// TwinCAT 3 PLC project Untitled1
// ProgramVersion: 3.1.4026.12
// libraries:
//   Tc2_Standard, * (Beckhoff Automation GmbH)
//   Tc2_System, * (Beckhoff Automation GmbH)
//   Tc3_Module, * (Beckhoff Automation GmbH)
//   VisuDialogs, * (System)
// project tree:
//   DUTs/ E_Bedrijfstoestand.TcDUT, E_OpenDichtKlepState.TcDUT, E_RegelingState.TcDUT, E_RegelschuifState.TcDUT, E_PompState.TcDUT, E_Besturingsmodus.TcDUT
//   / FB_AlarmHandler.TcPOU, GlobalTextList.TcGTLO, PlcTask.TcTTO, Visualization Manager.TcVMO (not stored)
//   POUs/ControlLayer/ FB_Inmalen.TcPOU, FB_Regelingen.TcPOU, FB_Uitlaten.TcPOU, FB_Uitmalen.TcPOU
//   POUs/DeviceLayer/ FB_OpenDichtKlep.TcPOU, FB_Pomp.TcPOU, FB_Regelschuif_DG.TcPOU, FB_Regelschuif_AFO.TcPOU, ITF_OpenDichtKlep.TcIO, ITF_Regelschuif.TcIO, ITF_Pomp.TcIO
//   POUs/FieldLayer/OpenDichtKlep/ FB_SimulatedDigIn.TcPOU, FB_SimulatedDigOut.TcPOU, ITF_DigIn.TcIO, ITF_DigOut.TcIO
//   POUs/FieldLayer/Pomp/ FB_simulatedpompdigin.TcPOU, FB_simulatedpompdigout.TcPOU, FB_simulatiepompangout.TcPOU, ITF_pompangout.TcIO, ITF_pompdigin.TcIO, ITF_pompdigout.TcIO
//   POUs/FieldLayer/Regelschuif_AFO/ FB_SimulatedAnaIn_AFO.TcPOU, FB_SimulatedDigOutClose_AFO.TcPOU, FB_SimulatedDigOutOpen_AFO.TcPOU, ITF_Schuif_AnaIn_AFO.TcIO, ITF_Schuif_DigOutClose_AFO.TcIO, ITF_Schuif_DigOutOpen_AFO.TcIO
//   POUs/FieldLayer/Regelschuif_DG_1/ FB_SimulatedIn_DG.TcPOU, FB_SimulatedOutClose_DG.TcPOU, FB_SimulatedOutOpen_DG.TcPOU, ITF_Regelschuif_In_DG.TcIO, ITF_Regelschuif_OutClose_DG.TcIO, ITF_Regelschuif_OutOpen_DG.TcIO
//   POUs/ MAIN.TcPOU
//   VISUs/ Visualization.TcVIS
// real-time tasks:
//   TASK PlcTask: cycle T#10ms, priority 20, ADS port 350

CONFIGURATION Untitled1
    RESOURCE PLC ON TwinCAT3
        TASK PlcTask(INTERVAL := T#10ms, PRIORITY := 20);
        PROGRAM MAIN WITH PlcTask : MAIN;
    END_RESOURCE
END_CONFIGURATION

// ---- DUTs/E_Bedrijfstoestand.TcDUT
{attribute 'qualified_only'}
{attribute 'strict'}
{attribute 'to_string'}
TYPE E_Bedrijfstoestand :
(
	off := 0,
	manual,
	auto
);
END_TYPE

// ---- DUTs/E_OpenDichtKlepState.TcDUT
{attribute 'qualified_only'}
{attribute 'strict'}
{attribute 'to_string'}
TYPE E_OpenDichtKlepState :
(
	closed := 0,
	open,
	closing,
	opening,
	error
);
END_TYPE

// ---- DUTs/E_RegelingState.TcDUT
{attribute 'qualified_only'}
{attribute 'strict'}
{attribute 'to_string'}
TYPE E_RegelingState :
(
	uit := 0,
	polderpeil,
	debiet
);
END_TYPE

// ---- DUTs/E_RegelschuifState.TcDUT
{attribute 'qualified_only'}
{attribute 'strict'}
{attribute 'to_string'}
TYPE E_RegelschuifState :
(
	standby := 0,
	opening,
	closing,
	error
);
END_TYPE

// ---- DUTs/E_PompState.TcDUT
{attribute 'qualified_only'}
{attribute 'strict'}
{attribute 'to_string'}
TYPE E_PompState :
(
	off := 0,
	on,
	optoeren,
	aftoeren,
	error
);
END_TYPE

// ---- DUTs/E_Besturingsmodus.TcDUT
{attribute 'qualified_only'}
{attribute 'strict'}
{attribute 'to_string'}
TYPE E_Besturingsmodus :
(
	uitlaten := 0,
	uitmalen,
	inmalen
);
END_TYPE

// ---- POUs/DeviceLayer/ITF_OpenDichtKlep.TcIO
INTERFACE ITF_OpenDichtKlep

METHOD Close : BOOL
VAR_INPUT
END_VAR
END_METHOD

METHOD Open : BOOL
VAR_INPUT
END_VAR
END_METHOD

PROPERTY StateKlep : E_OpenDichtKlepState
GET
END_GET
SET
END_SET
END_PROPERTY

END_INTERFACE

// ---- POUs/DeviceLayer/ITF_Regelschuif.TcIO
INTERFACE ITF_Regelschuif

PROPERTY ActueelPosition : SINT
GET
END_GET
SET
END_SET
END_PROPERTY

METHOD RegelSchuifGoTo : SINT
VAR_INPUT
	regelschuifdoel : SINT;
END_VAR
END_METHOD

PROPERTY StateRegelSchuif : E_RegelschuifState
GET
END_GET
SET
END_SET
END_PROPERTY

END_INTERFACE

// ---- POUs/DeviceLayer/ITF_Pomp.TcIO
INTERFACE ITF_Pomp

PROPERTY ActueelToerental : INT
GET
END_GET
SET
END_SET
END_PROPERTY

METHOD PompGoTo : INT
VAR_INPUT
	toerental : INT;
END_VAR
END_METHOD

PROPERTY StatePomp : E_PompState
GET
END_GET
SET
END_SET
END_PROPERTY

END_INTERFACE

// ---- POUs/FieldLayer/OpenDichtKlep/ITF_DigIn.TcIO
INTERFACE ITF_DigIn

METHOD get : BOOL
VAR_INPUT
END_VAR
END_METHOD

END_INTERFACE

// ---- POUs/FieldLayer/OpenDichtKlep/ITF_DigOut.TcIO
INTERFACE ITF_DigOut

METHOD set : BOOL
VAR_INPUT
	state : BOOL;
END_VAR
END_METHOD

END_INTERFACE

// ---- POUs/FieldLayer/Pomp/ITF_pompangout.TcIO
INTERFACE ITF_pompangout

METHOD set : INT
VAR_INPUT
		state : INT;
END_VAR
END_METHOD

END_INTERFACE

// ---- POUs/FieldLayer/Pomp/ITF_pompdigin.TcIO
INTERFACE ITF_pompdigin

METHOD get : bool
VAR_INPUT
	state : BOOL;
END_VAR
END_METHOD

END_INTERFACE

// ---- POUs/FieldLayer/Pomp/ITF_pompdigout.TcIO
INTERFACE ITF_pompdigout

METHOD set : bool
VAR_INPUT
	state : BOOL;
END_VAR
END_METHOD

END_INTERFACE

// ---- POUs/FieldLayer/Regelschuif_AFO/ITF_Schuif_AnaIn_AFO.TcIO
INTERFACE ITF_Schuif_AnaIn_AFO

METHOD get : SINT
VAR_INPUT
END_VAR
END_METHOD

END_INTERFACE

// ---- POUs/FieldLayer/Regelschuif_AFO/ITF_Schuif_DigOutClose_AFO.TcIO
INTERFACE ITF_Schuif_DigOutClose_AFO

METHOD set : BOOL
VAR_INPUT
	state : BOOL;	
END_VAR
END_METHOD

END_INTERFACE

// ---- POUs/FieldLayer/Regelschuif_AFO/ITF_Schuif_DigOutOpen_AFO.TcIO
INTERFACE ITF_Schuif_DigOutOpen_AFO

METHOD set : BOOL
VAR_INPUT
	state : BOOL;
END_VAR
END_METHOD

END_INTERFACE

// ---- POUs/FieldLayer/Regelschuif_DG_1/ITF_Regelschuif_In_DG.TcIO
INTERFACE ITF_Regelschuif_In_DG

METHOD get : SINT
VAR_INPUT
END_VAR
END_METHOD

END_INTERFACE

// ---- POUs/FieldLayer/Regelschuif_DG_1/ITF_Regelschuif_OutClose_DG.TcIO
INTERFACE ITF_Regelschuif_OutClose_DG

METHOD set : BOOL
VAR_INPUT
	state : BOOL;	
END_VAR
END_METHOD

END_INTERFACE

// ---- POUs/FieldLayer/Regelschuif_DG_1/ITF_Regelschuif_OutOpen_DG.TcIO
INTERFACE ITF_Regelschuif_OutOpen_DG

METHOD set : BOOL
VAR_INPUT
	state : BOOL;
END_VAR
END_METHOD

END_INTERFACE

// ---- POUs/MAIN.TcPOU
PROGRAM MAIN
VAR
	alarms  : FB_AlarmHandler;
	
	// Start digin digout van appeltjes
	digIn_V2012_1 : FB_SimulatedDigIn;
	digIn_V2012_2 : FB_SimulatedDigIn;
	digOut_V2012 : FB_SimulatedDigOut;
	
	digIn_V2014_1 : FB_SimulatedDigIn;
	digIn_V2014_2 : FB_SimulatedDigIn;
	digOut_V2014 : FB_SimulatedDigOut;
	
	digIn_V2021_1 : FB_SimulatedDigIn;
	digIn_V2021_2 : FB_SimulatedDigIn;
	digOut_V2021 : FB_SimulatedDigOut;
	
	digIn_V2023_1 : FB_SimulatedDigIn;
	digIn_V2023_2 : FB_SimulatedDigIn;
	digOut_V2023 : FB_SimulatedDigOut;
	
	digIn_V2024_1 : FB_SimulatedDigIn;
	digIn_V2024_2 : FB_SimulatedDigIn;
	digOut_V2024 : FB_SimulatedDigOut;
	
	digIn_V2025_1 : FB_SimulatedDigIn;
	digIn_V2025_2 : FB_SimulatedDigIn;
	digOut_V2025 : FB_SimulatedDigOut;
	
	digIn_V2026_1 : FB_SimulatedDigIn;
	digIn_V2026_2 : FB_SimulatedDigIn;
	digOut_V2026 : FB_SimulatedDigOut;
	// Einde digin digout van appeltjes
	
	// Start digin digout van AFO
	digOutOpeningV2013 : FB_SimulatedDigOutOpen_AFO;
	digOutClosingV2013 :FB_SimulatedDigOutClose_AFO;
	AnaInV2013 : FB_SimulatedAnaIn_AFO;
	
	digOutOpeningV2022 : FB_SimulatedDigOutOpen_AFO;
	digOutClosingV2022 :FB_SimulatedDigOutClose_AFO;
	AnaInV2022 : FB_SimulatedAnaIn_AFO;
	
	AFOTarget : SINT := 20; 
	AFOTarget2 : SINT; 
	// Einde digin digout van AFO

	//DG
	OutOpeningV2013 : FB_SimulatedOutOpen_DG;
	OutClosingV2013 :FB_SimulatedOutClose_DG;
	InV2013 : FB_SimulatedIn_DG;
	
	OutOpeningV2022 : FB_SimulatedOutOpen_DG;
	OutClosingV2022 :FB_SimulatedOutClose_DG;
	InV2022 : FB_SimulatedIn_DG;
	//DG

	// Start digin digout van queens of harts
	digoutP2011 :FB_simulatedpompdigout;
	digoutP2021 :FB_simulatedpompdigout;
	diginP2011 : FB_simulatedpompdigin;
	diginP2021 : FB_simulatedpompdigin;
	AnaoutP2011 : FB_simulatiepompangout;
	AnaoutP2021 : FB_simulatiepompangout;
	
	
	// einde digin digout van queens of harts
	V2012 : FB_OpenDichtKlep(tag := 'V2012', DigInClosed := digIn_V2012_1, DigInOpened := digIn_V2012_2, DigOut := digOut_V2012);
	V2014 : FB_OpenDichtKlep(tag := 'V2014', DigInClosed := digIn_V2014_1, DigInOpened := digIn_V2014_2, DigOut := digOut_V2014);
	V2021 : FB_OpenDichtKlep(tag := 'V2021', DigInClosed := digIn_V2021_1, DigInOpened := digIn_V2021_2, DigOut := digOut_V2021);
	V2023 : FB_OpenDichtKlep(tag := 'V2023', DigInClosed := digIn_V2023_1, DigInOpened := digIn_V2023_2, DigOut := digOut_V2023);
	V2024 : FB_OpenDichtKlep(tag := 'V2024', DigInClosed := digIn_V2024_1, DigInOpened := digIn_V2024_2, DigOut := digOut_V2024);  
	V2025 : FB_OpenDichtKlep(tag := 'V2025', DigInClosed := digIn_V2025_1, DigInOpened := digIn_V2025_2, DigOut := digOut_V2025);  
	V2026 : FB_OpenDichtKlep(tag := 'V2026', DigInClosed := digIn_V2026_1, DigInOpened := digIn_V2026_2, DigOut := digOut_V2026);  
	
	V2013_AFO : FB_Regelschuif_AFO(tag := 'V2013', DigOutOpening := digOutOpeningV2013, DigOutClosing := digOutClosingV2013, AnaInPosition := AnaInV2013);
	V2022_AFO : FB_Regelschuif_AFO(tag := 'V2022', DigOutOpening := digOutOpeningV2022, DigOutClosing := digOutClosingV2022, AnaInPosition := AnaInV2022);
	
	V2013_DG : FB_Regelschuif_DG(tag := 'V2013', OutputOpen := OutOpeningV2013, OutputClose := OutClosingV2013, SchuifInput := InV2013);
	V2022_DG : FB_Regelschuif_DG(tag := 'V2022', OutputOpen := OutOpeningV2022, OutputClose := OutClosingV2022, SchuifInput := InV2022);
	
	P2011 : FB_Pomp(tag:= 'P2011',DigOutOn:=digoutP2011,Diginon:=diginP2011, Anaouttoerental:=AnaoutP2011);
	P2021 : FB_Pomp(tag:= 'P2021',DigOutOn:=digoutP2021,Diginon:=diginP2021, Anaouttoerental:=AnaoutP2021);
	
	Regelingen : FB_Regelingen;
	
	ControllerInmalen : FB_Inmalen(OpenDichtKlepV2012 := V2012,
								   OpenDichtKlepV2014 := V2014,
								   OpenDichtKlepV2021 := V2021, 
								   OpenDichtKlepV2023 := V2023, 
								   OpenDichtKlepV2024 := V2024,
								   OpenDichtKlepV2025 := V2025,
								   OpenDichtKlepV2026 := V2026,
								   RegelschuifV2013_AFO := V2013_AFO,
								   RegelschuifV2022_AFO := V2022_AFO,
								   RegelschuifV2013_DG := V2013_DG,
								   RegelschuifV2022_DG := V2022_DG,
								   PompP2011 := P2011,
								   PompP2021 := P2021 );
								   
	ControllerUitmalen : FB_Uitmalen(OpenDichtKlepV2012 := V2012,
								   OpenDichtKlepV2014 := V2014,
								   OpenDichtKlepV2021 := V2021, 
								   OpenDichtKlepV2023 := V2023, 
								   OpenDichtKlepV2024 := V2024,
								   OpenDichtKlepV2025 := V2025,
								   OpenDichtKlepV2026 := V2026,
								   RegelschuifV2013_AFO := V2013_AFO,
								   RegelschuifV2022_AFO := V2022_AFO,
								   RegelschuifV2013_DG := V2013_DG,
								   RegelschuifV2022_DG := V2022_DG,
								   PompP2021 := P2021,
								   PompP2011 := P2011 );
								   
	ControllerUitlaten: FB_Uitlaten(OpenDichtKlepV2012:= V2012,
									OpenDichtKlepV2021:=V2021,
									OpenDichtKlepV2023:=V2023,
									OpenDichtKlepV2024:=V2024,
									V2013_DG:=V2013_DG,
									V2022_DG:=V2022_DG,
									V2013_AFO:=V2013_AFO,
									V2022_AFO:=V2022_AFO,
									Pomp2011:= P2011,
									Pomp2021:= P2021);					   
	ManToerental2011: INT;
	ManToerental2021: INT;
	
	ManKlepstand2013_DG: SINT;
	ManKlepstand2022_DG: SINT;
END_VAR

digIn_V2012_1();
digIn_V2012_2();
digOut_V2012();

digIn_V2021_1();
digIn_V2021_2();
digOut_V2021();

digIn_V2023_1();
digIn_V2023_2();
digOut_V2023();

digIn_V2024_1();
digIn_V2024_2();
digOut_V2024();

digIn_V2025_1();
digIn_V2025_2();
digOut_V2025();

digIn_V2026_1();
digIn_V2026_2();
digOut_V2026();

digIn_V2014_1();
digIn_V2014_2();
digOut_V2014();

V2012();
V2014();
V2021();
V2023();
V2024();
V2025();
V2026();
//End  function kleppen appeltjes

P2021();
P2011();
P2011.PompGoToManual(ManToerental2011);
P2021.PompGoToManual(ManToerental2021);


Regelingen ();
ControllerInmalen ();
ControllerUitmalen ();
ControllerUitlaten();

//AFO
digOutOpeningV2013();
digOutClosingV2013();
AnaInV2013();
V2013_AFO();
V2013_AFO.RegelSchuifGoTo(AFOTarget); // voor handmatige test
digOutOpeningV2022();
digOutClosingV2022();
AnaInV2022();
V2022_AFO();
V2022_AFO.RegelSchuifGoTo(AFOTarget2); // voor handmatige test

//DG
V2013_DG();
V2013_DG.RegelSchuifGoToManual(ManKlepstand2013_DG);
V2022_DG();
V2022_DG.RegelSchuifGoToManual(ManKlepstand2022_DG);

END_PROGRAM

// ---- FB_AlarmHandler.TcPOU
FUNCTION_BLOCK FB_AlarmHandler
VAR
END_VAR

METHOD Append : BOOL
VAR_INPUT
	tag : STRING;
	msg : STRING;
END_VAR
VAR
	str : STRING;
END_VAR
str := CONCAT(tag, ': ');
str := CONCAT(str, msg);
ADSLOGSTR(msgCtrlMask := ADSLOG_MSGTYPE_WARN OR ADSLOG_MSGTYPE_MSGBOX, msgFmtStr := '%s!', strArg := str);
END_METHOD

END_FUNCTION_BLOCK

// ---- POUs/FieldLayer/OpenDichtKlep/FB_SimulatedDigIn.TcPOU
FUNCTION_BLOCK FB_SimulatedDigIn IMPLEMENTS ITF_DigIn
VAR
	internalState : BOOL;
END_VAR

METHOD get : BOOL
VAR_INPUT
END_VAR
get := internalState;
END_METHOD

END_FUNCTION_BLOCK

// ---- POUs/FieldLayer/OpenDichtKlep/FB_SimulatedDigOut.TcPOU
FUNCTION_BLOCK FB_SimulatedDigOut IMPLEMENTS ITF_DigOut
VAR
	internalState : BOOL := FALSE;
END_VAR

METHOD set : BOOL
VAR_INPUT
	state : BOOL;
END_VAR
internalState := state;
END_METHOD

END_FUNCTION_BLOCK

// ---- POUs/FieldLayer/Regelschuif_AFO/FB_SimulatedDigOutOpen_AFO.TcPOU
FUNCTION_BLOCK FB_SimulatedDigOutOpen_AFO IMPLEMENTS ITF_Schuif_DigOutOpen_AFO
VAR
	internalState : BOOL := FALSE;
END_VAR

METHOD set : BOOL
VAR_INPUT
	state : BOOL;
END_VAR
internalState := state;
END_METHOD

END_FUNCTION_BLOCK

// ---- POUs/FieldLayer/Regelschuif_AFO/FB_SimulatedDigOutClose_AFO.TcPOU
FUNCTION_BLOCK FB_SimulatedDigOutClose_AFO IMPLEMENTS ITF_Schuif_DigOutClose_AFO
VAR
	internalState : BOOL := FALSE;
END_VAR

{warning 'Add method implementation '}
METHOD set : BOOL
VAR_INPUT
	state : BOOL;
END_VAR
internalState := state;
END_METHOD

END_FUNCTION_BLOCK

// ---- POUs/FieldLayer/Regelschuif_AFO/FB_SimulatedAnaIn_AFO.TcPOU
FUNCTION_BLOCK FB_SimulatedAnaIn_AFO IMPLEMENTS ITF_Schuif_AnaIn_AFO

VAR
	internalState : sint;
END_VAR

{warning 'Add method implementation '}
METHOD get : SINT
get := internalState;
END_METHOD

END_FUNCTION_BLOCK

// ---- POUs/FieldLayer/Regelschuif_DG_1/FB_SimulatedOutOpen_DG.TcPOU
FUNCTION_BLOCK FB_SimulatedOutOpen_DG IMPLEMENTS ITF_Regelschuif_OutOpen_DG
VAR
	internalState : BOOL := FALSE;
END_VAR

METHOD set : BOOL
VAR_INPUT
	state : BOOL;
END_VAR
internalState := state;
END_METHOD

END_FUNCTION_BLOCK

// ---- POUs/FieldLayer/Regelschuif_DG_1/FB_SimulatedOutClose_DG.TcPOU
FUNCTION_BLOCK FB_SimulatedOutClose_DG IMPLEMENTS ITF_Regelschuif_OutClose_DG
VAR
	internalState : BOOL := FALSE;
END_VAR

{warning 'Add method implementation '}
METHOD set : BOOL
VAR_INPUT
	state : BOOL;
END_VAR
internalState := state;
END_METHOD

END_FUNCTION_BLOCK

// ---- POUs/FieldLayer/Regelschuif_DG_1/FB_SimulatedIn_DG.TcPOU
FUNCTION_BLOCK FB_SimulatedIn_DG IMPLEMENTS ITF_Regelschuif_IN_DG

VAR
	internalState : sint;
END_VAR

{warning 'Add method implementation '}
METHOD get : SINT
get := internalState;
END_METHOD

END_FUNCTION_BLOCK

// ---- POUs/FieldLayer/Pomp/FB_simulatedpompdigout.TcPOU
FUNCTION_BLOCK FB_simulatedpompdigout IMPLEMENTS ITF_pompdigout
VAR
	internalState:BOOL;
END_VAR

{warning 'Add method implementation '}
METHOD set : BOOL
VAR_INPUT
	state	: BOOL;
END_VAR
internalState := state;
END_METHOD

END_FUNCTION_BLOCK

// ---- POUs/FieldLayer/Pomp/FB_simulatedpompdigin.TcPOU
FUNCTION_BLOCK FB_simulatedpompdigin IMPLEMENTS ITF_pompdigin
VAR
	internalState : bool;
END_VAR

{warning 'Add method implementation '}
METHOD get : BOOL
VAR_INPUT
	state	: BOOL;
END_VAR
get := internalState;
END_METHOD

END_FUNCTION_BLOCK

// ---- POUs/FieldLayer/Pomp/FB_simulatiepompangout.TcPOU
FUNCTION_BLOCK FB_simulatiepompangout IMPLEMENTS ITF_pompangout

VAR
		internalState : int;
END_VAR

METHOD set : INT
VAR_INPUT
	state	: INT;
END_VAR
internalState := state;
END_METHOD

END_FUNCTION_BLOCK

// ---- POUs/DeviceLayer/FB_OpenDichtKlep.TcPOU
FUNCTION_BLOCK FB_OpenDichtKlep IMPLEMENTS ITF_OpenDichtKlep
VAR
    tagName : STRING;
    inputOpen : ITF_DigIn;
	inputClosed : ITF_DigIn;
	output : ITF_DigOut;
	
	feedbackOpen : BOOL := FALSE;
	feedbackClosed : BOOL := FALSE;
	feedbackError : BOOL := FALSE;
	
	manOpen : BOOL := FALSE;
	manClose : BOOL := FALSE;

	currentMode : E_Bedrijfstoestand := E_Bedrijfstoestand.off;
	currentState : E_OpenDichtKlepState := E_OpenDichtKlepState.closed;
	expectedState : E_OpenDichtKlepState := E_OpenDichtKlepState.closed;
	
	timeOut : TON;
	errorTrigger : R_TRIG;
	

END_VAR

//check if currentmode = off and set klep closed
IF currentMode = E_Bedrijfstoestand.off THEN
	output.set(FALSE);
	expectedState := E_OpenDichtKlepState.closed;
END_IF

//check if currentmode = manual and give klep a state
IF currentMode = E_Bedrijfstoestand.manual THEN
	IF manOpen THEN
		openManual();
		manOpen:= FALSE;
	END_IF
	IF manClose THEN
		closeManual();
		manClose:= FALSE;
	END_IF
END_IF

//control witch feedback button in pressed
feedbackOpen := inputOpen.get() AND NOT inputClosed.get();
feedbackClosed := inputClosed.get() AND NOT inputOpen.get();
feedbackError := inputClosed.get() AND inputOpen.get();

//set timer for error
timeOut(IN := NOT(expectedState = currentState), PT := T#5S);
errorTrigger(CLK := (timeOut.Q OR feedbackError));

//check if error is active
IF errorTrigger.Q THEN
	currentState := E_OpenDichtKlepState.error;
	main.alarms.append(tag := tagName, msg := 'Klepstoring gedetecteerd');
END_IF

//set state of klep based on feedback buttons
IF feedbackClosed THEN
	currentState := E_OpenDichtKlepState.closed;
ELSIF NOT(currentState = E_OpenDichtKlepState.error) AND expectedState = E_OpenDichtKlepState.closed THEN
	currentState := E_OpenDichtKlepState.closing;
ELSIF feedbackOpen THEN
	currentState := E_OpenDichtKlepState.open;
ELSIF NOT(currentState = E_OpenDichtKlepState.error)AND expectedState = E_OpenDichtKlepState.open THEN
	currentState := E_OpenDichtKlepState.opening;
END_IF

METHOD close : BOOL
VAR_INPUT
END_VAR
IF currentMode = E_Bedrijfstoestand.auto THEN
	output.set(FALSE);
	expectedState := E_OpenDichtKlepState.closed;
	close := TRUE;
ELSE
	close := FALSE;
END_IF
END_METHOD

METHOD closeManual : BOOL
VAR_INPUT
END_VAR
IF currentMode = E_Bedrijfstoestand.manual THEN
	output.set(FALSE);
	expectedState := E_OpenDichtKlepState.closed;
	closeManual := TRUE;
ELSE
	closeManual := FALSE;
END_IF
END_METHOD

METHOD FB_init : BOOL
VAR_INPUT
	bInitRetains : BOOL; // if TRUE, the retain variables are initialized (warm start / cold start)
	bInCopyCode : BOOL;  // if TRUE, the instance afterwards gets moved into the copy code (online change)
	tag : STRING;
	DigInClosed : ITF_DigIn;
	DigInOpened : ITF_DigIn;
	DigOut : ITF_DigOut;
END_VAR
tagname := tag;
inputClosed := DigInClosed;
inputOpen := DigInOpened;
output := DigOut;
END_METHOD

METHOD open : BOOL
VAR_INPUT
END_VAR
IF currentMode = E_Bedrijfstoestand.auto THEN
	output.set(TRUE);
	expectedState := E_OpenDichtKlepState.open;
	open := TRUE;
ELSE
	open := FALSE;
END_IF
END_METHOD

METHOD openManual : BOOL
VAR_INPUT
END_VAR
IF currentMode = E_Bedrijfstoestand.manual THEN
	output.set(TRUE);
	expectedState := E_OpenDichtKlepState.open;
	openManual := TRUE;
ELSE
	openManual := FALSE;
END_IF
END_METHOD

PROPERTY StateKlep : E_OpenDichtKlepState
GET
StateKlep := currentState;
END_GET
SET
END_SET
END_PROPERTY

END_FUNCTION_BLOCK

// ---- POUs/DeviceLayer/FB_Regelschuif_AFO.TcPOU
FUNCTION_BLOCK FB_Regelschuif_AFO IMPLEMENTS ITF_Regelschuif
VAR
	tagName : STRING;
	outputOpen : ITF_Schuif_DigOutOpen_AFO;
	outputClose : ITF_Schuif_DigOutClose_AFO;
	inputPosition : ITF_Schuif_AnaIn_AFO;

	currentMode : E_Bedrijfstoestand := E_Bedrijfstoestand.off;
	currentState : E_RegelschuifState := E_RegelschuifState.standby;
	expectedState : E_RegelschuifState := E_RegelschuifState.standby;
	
	feedbackPosition : SINT;
	
	timeOut : TON;
	errorTrigger : R_TRIG;
	positie : SINT;
	secondTimerRun : BOOL;
	secondTimerTrigger : R_TRIG;
	
	timerrunt: BOOL:=1;
	waitExtraMinute: BOOL;
	minuteTimer : TON;
	doubleMinuteTimer : TON;
	secondTimer : TON;
	
	veranderingsMargeError : SINT := 3;
	OldPosition: SINT;
	regelschuifMargin: SINT := 3;
END_VAR

// Als de mode is uit dan worden de outputs false geset 
IF currentMode = E_Bedrijfstoestand.off THEN
	outputOpen.set(FALSE);
	outputClose.set(FALSE);
END_IF

// De feedback positie staat hiet zodat we de waardes kunnen veranderen
feedbackPosition := inputPosition.get();
ActueelPosition := inputPosition.get();

// Dit is de timer om te checken of er een error moet zijn 
timeOut(IN :=(StateRegelSchuif <> E_RegelschuifState.standby) AND NOT timeOut.Q, PT := T#30S);
errorTrigger(CLK := timeOut.Q);

IF errorTrigger.Q THEN
	IF (ActueelPosition < (OldPosition + veranderingsMargeError)) AND StateRegelSchuif = E_RegelschuifState.opening THEN
		StateRegelSchuif := E_RegelschuifState.error;
		main.alarms.append(tag := tagName, msg := 'Schuifstoring gedetecteerd, te langzaam openen');
	END_IF
	IF (ActueelPosition > (OldPosition - veranderingsMargeError)) AND StateRegelSchuif = E_RegelschuifState.closing THEN
		StateRegelSchuif := E_RegelschuifState.error;
		main.alarms.append(tag := tagName, msg := 'Schuifstoring gedetecteerd, te langzaam sluiten');
	END_IF
	IF StateRegelSchuif = E_RegelschuifState.error AND (ActueelPosition > (OldPosition + veranderingsMargeError)) THEN
		StateRegelSchuif := E_RegelschuifState.opening;
		ELSIF StateRegelSchuif = E_RegelschuifState.error AND (ActueelPosition < (OldPosition - veranderingsMargeError)) THEN
			StateRegelSchuif := E_RegelschuifState.closing;
	END_IF
	OldPosition := ActueelPosition;
END_IF

expectedState := StateRegelSchuif;

PROPERTY ActueelPosition : SINT
GET
ActueelPosition := feedbackPosition;
END_GET
SET
feedbackPosition := ActueelPosition;
END_SET
END_PROPERTY

//FB_Init is always available implicitly and it is used primarily for initialization.
//The return value is not evaluated. For a specific influence, you can also declare the
//methods explicitly and provide additional code there with the standard initialization
//code. You can evaluate the return value.
METHOD FB_Init: BOOL
VAR_INPUT
    bInitRetains: BOOL; // TRUE: the retain variables are initialized (reset warm / reset cold)
    bInCopyCode: BOOL;  // TRUE: the instance will be copied to the copy code afterward (online change)   
	tag : STRING;
	DigOutOpening : ITF_Schuif_DigOutOpen_AFO;
	DigOutClosing : ITF_Schuif_DigOutClose_AFO;
	AnaInPosition : ITF_Schuif_AnaIn_AFO;
END_VAR
tagname := tag;
outputOpen := DigOutOpening;
outputClose := DigOutClosing;
inputPosition := AnaInPosition;
END_METHOD

METHOD RegelSchuifGoTo : SINT
VAR	
	checkPositions : BOOL;
	currentstatet: E_RegelschuifState;
	secondTriggerTrigger: BOOL;
END_VAR
VAR_INPUT
	regelschuifdoel : SINT;
END_VAR
minuteTimer(IN:= timerrunt,PT:= T#10S);
doubleMinuteTimer(IN:= waitExtraMinute,PT:= T#10S); // tweede timer om een extra minuut te wachten na pulse maar niet langer te wachten met scannen

// dit is zodat het gefaseerd gaat een pulse per sec sturen
secondTimer(IN:= secondTimerRun,PT:= T#2S); // pulse lengte langer ivm testen

IF currentMode = E_Bedrijfstoestand.off THEN
	regelschuifdoel := ActueelPosition;
END_IF

IF minuteTimer.Q THEN
	
	IF ActueelPosition >= (regelschuifdoel - regelschuifMargin) AND ActueelPosition <= (regelschuifdoel + regelschuifMargin) THEN // huidige positie is correct binnen marge
		StateRegelSchuif := E_RegelschuifState.standby;
		outputOpen.set(FALSE); // set outputs naar 0 als extra backup
		outputClose.set(FALSE);
	
	END_IF
	
	IF ActueelPosition > (regelschuifdoel + regelschuifMargin) AND waitExtraMinute = FALSE THEN // huidige positie is te hoog
		IF stateRegelschuif <> E_RegelschuifState.error THEN
			StateRegelSchuif := E_RegelschuifState.closing;
		END_IF
		// voor de pulse		
		outputOpen.set(FALSE);
		outputClose.set(TRUE);
		secondTimerRun := TRUE; // start pulse time
		waitExtraMinute := TRUE; // wacht een minuut extra als er een pulse is gestuurd
	END_IF

	IF ActueelPosition < (regelschuifdoel - regelschuifMargin) AND waitExtraMinute = FALSE THEN // huidige positie is te laag
		IF stateRegelschuif <> E_RegelschuifState.error THEN
			StateRegelSchuif := E_RegelschuifState.opening;
		END_IF
		// voor de pulse
		outputClose.set(FALSE);
		outputOpen.set(TRUE);
		secondTimerRun := TRUE; // start pulse time
		waitExtraMinute := TRUE;
	END_IF
	timerrunt := 0; // reset timer
ELSIF waitExtraMinute = FALSE OR doubleMinuteTimer.Q THEN 
	waitExtraMinute := FALSE;
	timerrunt := 1; //reser reset timer
END_IF

// pulse timer structuur
IF secondTimer.Q THEN
	outputClose.set(FALSE);
	outputOpen.set(FALSE);
	secondTimerRun := FALSE;
END_IF

positie := regelschuifdoel;
END_METHOD

PROPERTY StateRegelSchuif : E_RegelschuifState
GET
StateRegelschuif := currentState;
END_GET
SET
currentstate:= StateRegelSchuif;
END_SET
END_PROPERTY

END_FUNCTION_BLOCK

// ---- POUs/DeviceLayer/FB_Regelschuif_DG.TcPOU
FUNCTION_BLOCK FB_Regelschuif_DG IMPLEMENTS ITF_Regelschuif
VAR
	TagName: STRING;
	
	OpenSchuif: ITF_Regelschuif_OutOpen_DG;
	SluitSchuif: ITF_Regelschuif_OutClose_DG;
	InputSchuif: ITF_Regelschuif_In_DG;
	
	CurrentMode: E_Bedrijfstoestand:= E_Bedrijfstoestand.off;
	currentState : E_RegelschuifState := E_RegelschuifState.standby;
	expectedState : E_RegelschuifState := E_RegelschuifState.standby;
	
	feedbackposition: SINT;
	VorigePosition: SINT;
	Marge : SINT := 2;
	schuifverandering: SINT:= 1;
	Doelschuif: SINT;
	DoelschuifAuto : SINT;
	VorigDoel: SINT;
	
	PulseTimer: TON;
	StartPulse: BOOL;
	Pulsetrigger: R_TRIG;
	
	OptelTimer: TON;
	StartOptel: BOOL;
	
	error_Trigger: R_TRIG;
	ErrorTimer: TON;
	SchuifsturingOpen: BOOL;
	SchuifsturingSluit: BOOL;
	SchuifStandby: BOOL;
END_VAR

//Als de schuif uit staat stopt de regelschuif met openen of sluiten
IF CurrentMode = E_Bedrijfstoestand.off THEN
	Currentstate:= E_Regelschuifstate.standby;
END_IF

//De actuele positie van de schuif wordt geupdate
ActueelPosition:= Feedbackposition;

ErrorTimer(IN:= Currentstate <> E_Regelschuifstate.standby AND NOT ErrorTimer.Q ,PT:= T#5S);
error_Trigger(CLK:= ErrorTimer.Q);

PulseTimer(IN:=StartPulse AND NOT PulseTimer.Q ,PT:= T#10S);
Pulsetrigger(CLK:= Pulsetimer.Q);
IF (Currentmode <> E_Bedrijfstoestand.off) AND NOT Pulsetimer.Q THEN
	Startpulse:= 1;
END_IF

IF Currentmode = E_Bedrijfstoestand.off THEN
	SchuifsturingOpen := FALSE;
	SchuifsturingSluit := FALSE;
	Openschuif.set(FALSE);
	SluitSchuif.set(FALSE);
END_IF

IF (Pulsetrigger.Q) OR ((Doelschuif <> Vorigdoel)
AND CurrentMode = E_Bedrijfstoestand.manual) THEN
	Startpulse:= 0;
	IF (Doelschuif < Feedbackposition) THEN
		SchuifsturingOpen := FALSE;
		SchuifsturingSluit := TRUE;
	END_IF	
	IF (Doelschuif > Feedbackposition) THEN
		SchuifsturingOpen := TRUE;
		SchuifsturingSluit := FALSE;
	END_IF
	StartPulse:= 1;
	Vorigdoel:= Doelschuif;
END_IF

IF Feedbackposition = 100 OR Feedbackposition = 0 THEN;
	Currentstate := E_RegelschuifState.standby;
	Schuifsturing();
ELSIF (Doelschuif < Feedbackposition) THEN
	Currentstate := E_RegelschuifState.closing;
ELSIF (Doelschuif > Feedbackposition) THEN
	Currentstate := E_RegelschuifState.opening;
ELSIF (DoelschuifAuto < Feedbackposition) THEN
	Currentstate := E_RegelschuifState.closing;
ELSIF (DoelschuifAuto > Feedbackposition) THEN
	Currentstate := E_RegelschuifState.opening;
END_IF

IF SchuifsturingSluit OR SchuifsturingOpen THEN
	Schuifsturing();
END_IF


IF (Pulsetrigger.Q)
AND CurrentMode = E_Bedrijfstoestand.auto THEN
	Startpulse:= 0;
	IF (DoelschuifAuto < Feedbackposition) THEN
		SchuifsturingOpen := FALSE;
		SchuifsturingSluit := TRUE;
	END_IF	
	IF (DoelschuifAuto > Feedbackposition) THEN
		SchuifsturingOpen := TRUE;
		SchuifsturingSluit := FALSE;
	END_IF
	StartPulse:= 1;
END_IF

PROPERTY ActueelPosition : SINT
GET
END_GET
SET
END_SET
END_PROPERTY

METHOD FB_init : BOOL
VAR_INPUT
	bInitRetains : BOOL; // if TRUE, the retain variables are initialized (warm start / cold start)
	bInCopyCode : BOOL;  // if TRUE, the instance afterwards gets moved into the copy code (online change)
	
	tag: STRING;
	SchuifInput: ITF_Regelschuif_In_DG;
	OutputOpen: ITF_Regelschuif_OutOpen_DG;
	OutputClose: ITF_Regelschuif_OutClose_DG;
	
END_VAR
TagName:= tag;
InputSchuif := SchuifInput;
OpenSchuif := OutputOpen;
SluitSchuif := OutputClose;
END_METHOD

METHOD RegelSchuifGoTo : SINT

VAR_INPUT
	regelschuifdoel: SINT;
END_VAR
IF currentmode = E_Bedrijfstoestand.auto THEN
	DoelschuifAuto :=regelschuifdoel;
END_IF;





	//Zorgt ervoor dat de schuif stopt met bewegen als hij wordt uitgeschakeld
	IF CurrentMode = E_Bedrijfstoestand.off THEN
	regelschuifdoel := Feedbackposition;
	END_IF
END_METHOD

METHOD RegelschuifGoToManual : SINT

VAR_INPUT
	regelschuifdoelManual: SINT;
END_VAR
IF currentmode = E_Bedrijfstoestand.manual THEN
	Doelschuif:=regelschuifdoelManual;
END_IF;




	//Zorgt ervoor dat de schuif stopt met bewegen als hij wordt uitgeschakeld
	IF CurrentMode = E_Bedrijfstoestand.off THEN
	regelschuifdoelManual := Feedbackposition;
	END_IF
END_METHOD

METHOD Schuifsturing : SINT
VAR
END_VAR
Opteltimer(IN:= StartOptel, PT:= T#500MS);

IF Currentstate = E_RegelschuifState.standby THEN
		Openschuif.set(FALSE);
		Sluitschuif.set(FALSE);
END_IF
	//De regelschuif wordt geopend
	IF SchuifsturingOpen AND Feedbackposition <= 99 THEN
		Startoptel:= 1;
		OpenSchuif.set(TRUE);
		SluitSchuif.set(FALSE);
		IF Opteltimer.Q THEN
		Feedbackposition := Feedbackposition + schuifverandering;
		Startoptel:= 0;
		END_IF
	END_IF

	//De regelschuif wordt gesloten
	IF SchuifsturingSluit AND Feedbackposition >= 1 THEN
		Startoptel:= 1;
		Openschuif.set(FALSE);
		SluitSchuif.set(TRUE);
		IF Opteltimer.Q THEN
		Feedbackposition := Feedbackposition - schuifverandering;
		startoptel:= 0;
		END_IF
	END_IF
END_METHOD

PROPERTY StateRegelschuif : E_RegelschuifState
GET
END_GET
SET
END_SET
END_PROPERTY

END_FUNCTION_BLOCK

// ---- POUs/DeviceLayer/FB_Pomp.TcPOU
FUNCTION_BLOCK FB_Pomp IMPLEMENTS ITF_Pomp
VAR
	InternalToerental : INT; // Internal variable for current speed
 	InternalState : E_PompState;    // Internal variable for pump state
	InternalToerental2 : INT; // Internal variable for current speed
	globaaldoeltoerental : INT; //global variable for doel speed
	
	timeroptoeren : TON;
	timerloopt : BOOL := TRUE;
	optoerentimer : TIME := T#1M;
	
	visvriendelijkactief : BOOL:=visvriendelijkopstartenactief;
	
	//visvriendelijk timer
	timervisvriendelijktijd : TIME := T#3M;
	timervisvriendelijk : TON;
	bezig_visvriendelijkopstarten : BOOL := FALSE;
	
	tagName : STRING;
	outputpompon : ITF_pompdigout;
	inputpompon : ITF_pompdigin;
	outputtoerental : ITF_pompangout;
	
	timerpomperror: ton;
	timerpomperrortijd: TIME:=T#20S;
	noodstop:BOOL;
	
	Bedrijftoestand: E_Bedrijfstoestand := E_bedrijfstoestand.auto;
	
	
END_VAR

IF bedrijftoestand = E_bedrijfstoestand.off THEN
	internaltoerental := 0;
	globaaldoeltoerental := 0;
END_IF

//visvriendelijk
visvriendelijk();

//outputs pomp
ActueelToerental:=InternalToerental;
outputtoerental.set(InternalToerental);
IF InternalToerental = 0 AND globaaldoeltoerental=0 THEN
	outputpompon.set(FALSE);
ELSIF globaaldoeltoerental>0 THEN
	outputpompon.set(TRUE);
END_IF
//inputs errorcheck
timerpomperror(in:=(  (NOT inputpompon.get(FALSE)) AND(globaaldoeltoerental>0 AND ActueelToerental>0)) OR(inputpompon.get(TRUE) AND ((InternalToerental = 0 AND globaaldoeltoerental=0) OR ActueelToerental=0)), PT:=timerpomperrortijd);
IF timerpomperror.Q THEN
	InternalState := E_PompState.error;
END_IF

//status pomp
IF (NOT timerpomperror.Q) THEN
	IF  (NOT inputpompon.get(FALSE)) AND ActueelToerental=0 THEN
		InternalState := E_pompstate.off;
	ELSIF inputpompon.get(TRUE) AND ActueelToerental<globaaldoeltoerental THEN
		InternalState := E_pompstate.optoeren;
	ELSIF inputpompon.get(TRUE) AND ActueelToerental>globaaldoeltoerental THEN
		InternalState := E_pompstate.aftoeren;
	ELSIF inputpompon.get(TRUE) AND ActueelToerental=globaaldoeltoerental THEN
		InternalState := E_pompstate.on;
	END_IF
END_IF

{warning 'Add property implementation'}
PROPERTY ActueelToerental : INT
GET
 ActueelToerental := InternalToerental;
END_GET
SET
    InternalToerental := ActueelToerental;
END_SET
END_PROPERTY

//FB_Init is always available implicitly and it is used primarily for initialization.
//The return value is not evaluated. For a specific influence, you can also declare the
//methods explicitly and provide additional code there with the standard initialization
//code. You can evaluate the return value.
METHOD FB_Init: BOOL
VAR_INPUT
    bInitRetains: BOOL; // TRUE: the retain variables are initialized (reset warm / reset cold)
    bInCopyCode: BOOL;  // TRUE: the instance will be copied to the copy code afterward (online change)   
	tag : STRING;
	DigOutOn : ITF_pompdigout;
	Diginon : ITF_pompdigin;
	Anaouttoerental : ITF_pompangout;
END_VAR
tagname := tag;
outputpompon := DigOutOn;
inputpompon := Diginon;
outputtoerental := Anaouttoerental;
END_METHOD

METHOD PompGoTo : INT
VAR_INPUT
	toerental	: INT;
END_VAR

VAR
	afnametoerental : INT :=20;
	toenamentoerental : INT :=20;
END_VAR
IF Bedrijftoestand = E_Bedrijfstoestand.auto THEN
timeroptoeren(IN := timerloopt, PT := optoerentimer);
globaaldoeltoerental:=toerental;
IF noodstop THEN
	InternalToerental:=0;
ELSIF timeroptoeren.Q AND NOT bezig_visvriendelijkopstarten THEN
	timerloopt := FALSE;
	IF (toerental <= InternalToerental+toenamentoerental) AND (toerental >= InternalToerental-afnametoerental) THEN
		IF toerental >20 OR TOERENTAL=0THEN	
		InternalToerental:= toerental;
		ELSIF TOERENTAL>0 THEN
			INTERNALTOERENTAL:=20;
		END_IF;
	ELSIF toerental > InternalToerental THEN
	InternalToerental := InternalToerental+toenamentoerental;
	ELSIF toerental < internaltoerental THEN
		internaltoerental := InternalToerental-afnametoerental;
	END_IF;
ELSE
	timerloopt:=TRUE;
END_IF
END_IF
END_METHOD

METHOD PompGoToManual : INT
VAR_INPUT
	toerental	: INT;
END_VAR

VAR
	afnametoerental : INT :=20;
	toenamentoerental : INT :=20;
END_VAR
IF Bedrijftoestand = E_Bedrijfstoestand.manual THEN
timeroptoeren(IN := timerloopt, PT := optoerentimer);
globaaldoeltoerental:=toerental;
IF noodstop THEN
	InternalToerental:=0;
ELSIF timeroptoeren.Q AND NOT bezig_visvriendelijkopstarten THEN
	timerloopt := FALSE;
	IF (toerental <= InternalToerental+toenamentoerental) AND (toerental >= InternalToerental-afnametoerental) THEN
		IF toerental >20 OR TOERENTAL=0THEN	
		InternalToerental:= toerental;
		ELSIF TOERENTAL>0 THEN
			INTERNALTOERENTAL:=20;
		END_IF;
	ELSIF toerental > InternalToerental THEN
	InternalToerental := InternalToerental+toenamentoerental;
	ELSIF toerental < internaltoerental THEN
		internaltoerental := InternalToerental-afnametoerental;
	END_IF;
ELSE
	timerloopt:=TRUE;
END_IF
END_IF
END_METHOD

{warning 'Add property implementation'}
PROPERTY StatePomp : E_PompState
GET
    StatePomp := InternalState;
END_GET
SET
    InternalState := StatePomp;
END_SET
END_PROPERTY

METHOD visvriendelijk : BOOL
VAR_INPUT
END_VAR
timervisvriendelijk(IN:= bezig_visvriendelijkopstarten, PT:= timervisvriendelijktijd);

IF visvriendelijkactief AND (StatePomp = E_PompState.off OR bezig_visvriendelijkopstarten) AND globaaldoeltoerental>0 THEN
	bezig_visvriendelijkopstarten:=TRUE;
END_IF
IF bezig_visvriendelijkopstarten=TRUE THEN
	IF timervisvriendelijk.Q THEN
		bezig_visvriendelijkopstarten:=FALSE;
	ELSE
		InternalToerental:=20;
	END_IF
END_IF
END_METHOD

PROPERTY visvriendelijkopstartenactief : bool
GET
visvriendelijkopstartenactief:=visvriendelijkactief;
END_GET
SET
visvriendelijkactief:=visvriendelijkopstartenactief;
END_SET
END_PROPERTY

END_FUNCTION_BLOCK

// ---- POUs/ControlLayer/FB_Regelingen.TcPOU
FUNCTION_BLOCK FB_Regelingen
VAR
	internalBesturingsMode : E_Besturingsmodus;
	internalRegelschuifStandV2013 : SINT;
	internalRegelschuifStandV2022 : SINT;
	internalToerentalP2011 : INT;
	internalToerentalP2021 : INT;
	toerntalP2011p : INT := 40;
	toerentalP2021p : INT := 70;
	regelschuifV2013: SINT:=90;
	regelschuifV2022: SINT:=30;
	b: E_Besturingsmodus;
END_VAR

internalToerentalP2011 := toerntalP2011p;
internalToerentalP2021 := toerentalP2021p;
internalRegelschuifStandV2013 :=regelschuifV2013;
internalRegelschuifStandV2022 :=regelschuifV2022;
internalBesturingsMode := b;

PROPERTY BestuurMode : E_Besturingsmodus
GET
BestuurMode := internalBesturingsMode;
END_GET
SET
internalBesturingsMode := BestuurMode ;
END_SET
END_PROPERTY

PROPERTY RegelschuifStandV2013 : SINT
GET
RegelschuifStandV2013 := internalRegelschuifStandV2013;
END_GET
SET
internalRegelschuifStandV2013 := RegelschuifStandV2013;
END_SET
END_PROPERTY

PROPERTY RegelschuifStandV2022 : SINT
GET
RegelschuifStandV2022 := internalRegelschuifStandV2022;
END_GET
SET
internalRegelschuifStandV2022 := RegelschuifStandV2022;
END_SET
END_PROPERTY

PROPERTY ToerentalP2011 : INT
GET
ToerentalP2011 := internalToerentalP2011;
END_GET
SET
internalToerentalP2011 := ToerentalP2011;
END_SET
END_PROPERTY

PROPERTY ToerentalP2021 : INT
GET
ToerentalP2021 := internalToerentalP2021;
END_GET
SET
internalToerentalP2021 := ToerentalP2021;
END_SET
END_PROPERTY

END_FUNCTION_BLOCK

// ---- POUs/ControlLayer/FB_Inmalen.TcPOU
FUNCTION_BLOCK FB_Inmalen
VAR
	CurrentModus : E_Besturingsmodus := E_Besturingsmodus.uitlaten;
	KlepV2012 : ITF_OpenDichtKlep;
	KlepV2014 : ITF_OpenDichtKlep;
	KlepV2021 : ITF_OpenDichtKlep;
	KlepV2023 : ITF_OpenDichtKlep;
	KlepV2024 : ITF_OpenDichtKlep;
	KlepV2025 : ITF_OpenDichtKlep;
	KlepV2026 : ITF_OpenDichtKlep;
	
	SchuifV2013_AFG : ITF_Regelschuif;
	SchuifV2022_AFG : ITF_Regelschuif;
	
	SchuifV2013_DG : ITF_Regelschuif;
	SchuifV2022_DG : ITF_Regelschuif;
	
	pomp2_P2011 : ITF_Pomp;
	pomp2_P2021 : ITF_Pomp;
	
	pompP2011 : INT;
	pompP2021 : INT;
	
	Ontluchtingsklep : BOOL := FALSE;
	
	firstround : BOOL := FALSE;
	
	timeOut : TON;
	trigger : R_TRIG;
	TimerOn : BOOL := FALSE;
	
	First : BOOL := FALSE;
	
	PompAan : BOOL := FALSE;
END_VAR

//set currentmode to actual mode
CurrentModus:= main.Regelingen.BestuurMode;

IF (CurrentModus = E_Besturingsmodus.uitlaten) OR (CurrentModus = E_Besturingsmodus.uitmalen) THEN
	firstround := FALSE;
	First := FALSE;
	PompAan := FALSE;
END_IF

//Start modus inmalen			
IF CurrentModus = E_Besturingsmodus.inmalen THEN
	
	IF First = FALSE THEN
	//set position kleppen
	KlepV2012.close();
	KlepV2014.close();
	KlepV2021.Close();
	KlepV2024.Close();
	KlepV2025.close();
	KlepV2026.close();
	First := TRUE;
	END_IF
	
	//set position regelschuiven
	SchuifV2013_AFG.RegelSchuifGoTo(0);
	SchuifV2013_DG.RegelSchuifGoTo(0);
	
	IF (KlepV2012.StateKlep = E_OpenDichtKlepState.closed AND
		KlepV2021.StateKlep = E_OpenDichtKlepState.closed AND
		KlepV2024.StateKlep = E_OpenDichtKlepState.closed AND
		KlepV2025.StateKlep = E_OpenDichtKlepState.closed AND
		KlepV2026.StateKlep = E_OpenDichtKlepState.closed AND
		SchuifV2013_AFG.StateRegelSchuif = E_RegelschuifState.standby AND
		SchuifV2013_DG.StateRegelSchuif = E_RegelschuifState.standby) THEN
		
		//set position kleppen and regelschuiven
		KlepV2023.Open();
		SchuifV2022_AFG.RegelSchuifGoTo(100);
		SchuifV2022_DG.RegelSchuifGoTo(100);
		
		IF (KlepV2023.StateKlep = E_OpenDichtKlepState.open AND
			SchuifV2022_AFG.StateRegelSchuif = E_RegelschuifState.standby AND
			SchuifV2022_DG.StateRegelSchuif = E_RegelschuifState.standby) THEN
			
			//Get toerental
			pompP2011 := main.Regelingen.ToerentalP2011;
			pompP2021 := main.Regelingen.ToerentalP2021;
			
			//Set pomp on or off with toerental from regelingen
			pomp2_P2011.PompGoTo(pompP2011);
			pomp2_P2021.PompGoTo(pompP2021);

			IF 	pomp2_P2021.StatePomp = E_PompState.on THEN
				PompAan := TRUE;
			END_IF
		END_IF	
	END_IF	
	//Ontluchtingsklep open and after 10 seconds closed only when 
	IF firstRound = FALSE AND PompAan = TRUE THEN
		KlepV2025.open();
		
		IF KlepV2025.StateKlep = E_OpenDichtKlepState.open THEN
			TimerOn := TRUE;
	
			IF trigger.Q THEN
				KlepV2025.close();
				firstround := TRUE;
				TimerOn := FALSE;
			END_IF
		END_IF
	END_IF
	//timer ontluchtingsklep
	timeOut(IN := TimerOn, PT := T#10S);
	trigger(CLK := (timeOut.Q));
END_IF

METHOD FB_init : BOOL
VAR_INPUT
	bInitRetains : BOOL; // if TRUE, the retain variables are initialized (warm start / cold start)
	bInCopyCode : BOOL;  // if TRUE, the instance afterwards gets moved into the copy code (online change)
	OpenDichtKlepV2012 : ITF_OpenDichtKlep; 
	OpenDichtKlepV2014 : ITF_OpenDichtKlep; 
	OpenDichtKlepV2021 : ITF_OpenDichtKlep; 
	OpenDichtKlepV2023 : ITF_OpenDichtKlep; 
	OpenDichtKlepV2024 : ITF_OpenDichtKlep;
	OpenDichtKlepV2025 : ITF_OpenDichtKlep; 
	OpenDichtKlepV2026 : ITF_OpenDichtKlep;  
	
	RegelschuifV2013_AFO : ITF_Regelschuif; 
	RegelschuifV2022_AFO : ITF_Regelschuif;
	
	RegelschuifV2013_DG : ITF_Regelschuif;
	RegelschuifV2022_DG : ITF_Regelschuif;
	
	PompP2011 : ITF_Pomp;
	PompP2021 : ITF_Pomp;
	
END_VAR
KlepV2012 := OpenDichtKlepV2012;
KlepV2014 := OpenDichtKlepV2014;
KlepV2021 := OpenDichtKlepV2021;
KlepV2023 := OpenDichtKlepV2023;
KlepV2024 := OpenDichtKlepV2024;
KlepV2025 := OpenDichtKlepV2025;
KlepV2026 := OpenDichtKlepV2026;

SchuifV2013_AFG := RegelschuifV2013_AFO;
SchuifV2022_AFG := RegelschuifV2022_AFO;
SchuifV2013_DG := RegelschuifV2013_DG;
SchuifV2022_DG := RegelschuifV2022_DG;

pomp2_P2011 := PompP2011;
pomp2_P2021 := PompP2021;
END_METHOD

END_FUNCTION_BLOCK

// ---- POUs/ControlLayer/FB_Uitmalen.TcPOU
FUNCTION_BLOCK FB_Uitmalen
VAR_INPUT
	
END_VAR
VAR_OUTPUT
END_VAR
VAR
	stap : INT :=1;
	
	KlepV2012 : ITF_OpenDichtKlep;
	KlepV2014 : ITF_OpenDichtKlep;
	KlepV2021 : ITF_OpenDichtKlep;
	KlepV2023 : ITF_OpenDichtKlep;
	KlepV2024 : ITF_OpenDichtKlep;
	KlepV2025 : ITF_OpenDichtKlep;
	KlepV2026 : ITF_OpenDichtKlep;
	
	
	SchuifV2013_AFG : ITF_Regelschuif;
	SchuifV2022_AFG : ITF_Regelschuif;
	
	SchuifV2013_DG : ITF_Regelschuif;
	SchuifV2022_DG : ITF_Regelschuif;
	
	Pomp1_P2011 : ITF_Pomp;
	pomp2_P2021 : ITF_Pomp;
	
	pompP2011:INT;
	pompP2021:INT;
	
	
	
	tijd: TIME := T#5s;
	timerOntluchtingsklepV2014: TON;
	timerOntluchtingsklepV2026: TON;
	triggerOntluchtingsklepV2026: R_TRIG;
	triggerOntluchtingsklepV2014: R_TRIG;
	
	EersteKeerV2014: BOOL := TRUE;
	EersteKeerV2026: BOOL := TRUE;
END_VAR

IF main.Regelingen.BestuurMode = E_Besturingsmodus.uitmalen THEN	
CASE stap OF
	1:
		Pomp1_P2011.PompGoTo(0);
		pomp2_P2021.PompGoTo(0);
		IF 0 = Pomp1_P2011.ActueelToerental  AND
		   E_POMPSTATE.off = Pomp1_P2011.StatePomp AND 
		   0 = pomp2_P2021.ActueelToerental  AND 
		   E_POMPSTATE.off = pomp2_P2021.StatePomp THEN
			stap := 2;
		END_IF
			
	2:
		SchuifV2013_AFG.RegelschuifGoTo(0);
		SchuifV2022_AFG.RegelschuifGoTo(0);
		KlepV2012.Open();
		KlepV2014.Close();
		KlepV2021.Open();
		KlepV2023.Close();
		KlepV2024.Open();
		KlepV2026.Close();
		IF 0 = SchuifV2013_AFG.ActueelPosition  AND 
		   E_RegelschuifState.standby = SchuifV2013_AFG.StateRegelschuif AND
		   0 = SchuifV2022_AFG.ActueelPosition  AND 
		   E_RegelschuifState.standby = SchuifV2022_AFG.StateRegelschuif AND 
		   E_OpenDichtKlepState.open = KlepV2012.StateKlep AND 
		   E_OpenDichtKlepState.closed = KlepV2014.StateKlep AND 
		   E_OpenDichtKlepState.open = KlepV2021.StateKlep AND
		   E_OpenDichtKlepState.closed = KlepV2023.StateKlep AND 
		   E_OpenDichtKlepState.open = KlepV2024.StateKlep  AND  
		   E_OpenDichtKlepState.closed = KlepV2026.StateKlep  THEN
			  stap := 3;
		END_IF
	3:
		pompP2011 := main.Regelingen.ToerentalP2011; // get toerental 11
		pompP2021 := main.Regelingen.ToerentalP2021; // get toerental 21
		pomp2_P2021.PompGoTo(pompP2021);//Set toerental 21
		Pomp1_P2011.PompGoTo(pompP2011); // set toerental 11
		
		
		IF  E_PompState.optoeren = Pomp1_P2011.StatePomp AND 
			EersteKeerV2014 = TRUE THEN // onluchtingklep p2011
				EersteKeerV2014 := FALSE;			
				KlepV2014.Open();
				timerOntluchtingsklepV2014 (IN:= E_OpenDichtKLepState.Open = KlepV2014.StateKlep, PT := tijd);
				triggerOntluchtingsklepV2014 (CLK := (timerOntluchtingsklepV2014.Q));
			IF triggerOntluchtingsklepV2014.Q  THEN
				KlepV2014.Close();
			END_IF
		END_IF
		
		IF  E_PompState.optoeren = pomp2_P2021.StatePomp AND 
			EersteKeerV2026 = TRUE THEN // ontluchtingsklep p2021
				EersteKeerV2026 := FALSE;
				KlepV2026.Open();
				timerOntluchtingsklepV2026 (IN:= E_OpenDichtKLepState.Open = KlepV2026.StateKlep, PT := tijd);
				triggerOntluchtingsklepV2026(CLK := (timerOntluchtingsklepV2026.Q));
				IF triggerOntluchtingsklepV2026.Q THEN
					KlepV2026.Close();
			END_IF
		END_IF
		
END_CASE
END_IF

//FB_Init is always available implicitly and it is used primarily for initialization.
//The return value is not evaluated. For a specific influence, you can also declare the
//methods explicitly and provide additional code there with the standard initialization
//code. You can evaluate the return value.
METHOD FB_Init: BOOL
VAR_INPUT
    bInitRetains: BOOL; // TRUE: the retain variables are initialized (reset warm / reset cold)
    bInCopyCode: BOOL;  // TRUE: the instance will be copied to the copy code afterward (online change)   
		OpenDichtKlepV2012: ITF_OpenDichtKlep;
	OpenDichtKlepV2014: ITF_OpenDichtKlep;
	OpenDichtKlepV2021: ITF_OpenDichtKlep;
	OpenDichtKlepV2023: ITF_OpenDichtKlep;
	OpenDichtKlepV2024: ITF_OpenDichtKlep;
	OpenDichtKlepV2025: ITF_OpenDichtKlep;
	OpenDichtKlepV2026: ITF_OpenDichtKlep;

	RegelschuifV2013_AFO: ITF_Regelschuif;
	RegelschuifV2022_AFO: ITF_Regelschuif;
	
	PompP2021: ITF_Pomp;
	PompP2011: ITF_Pomp;


	RegelschuifV2013_DG: ITF_Regelschuif;
	RegelschuifV2022_DG: ITF_Regelschuif;
END_VAR

	
KlepV2012 := OpenDichtKlepV2012;
KlepV2014 := OpenDichtKlepV2014;
KlepV2021 := OpenDichtKlepV2021;
KlepV2023 := OpenDichtKlepV2023;
KlepV2024 := OpenDichtKlepV2024;
KlepV2025 := OpenDichtKlepV2025;
KlepV2026 := OpenDichtKlepV2026;

SchuifV2013_AFG := RegelschuifV2013_AFO;
SchuifV2022_AFG := RegelschuifV2022_AFO;
SchuifV2013_DG := RegelschuifV2013_DG;
SchuifV2022_DG := RegelschuifV2022_DG;

pomp2_P2021 := PompP2021;
pomp1_p2011 := PompP2011;
END_METHOD

END_FUNCTION_BLOCK

// ---- POUs/ControlLayer/FB_Uitlaten.TcPOU
FUNCTION_BLOCK FB_Uitlaten
VAR
	Besturing: E_Besturingsmodus;

	PompStatus11 : ITF_Pomp;
	PompStatus21 : ITF_Pomp;
	
	KlepV2012 : ITF_OpenDichtKlep;
	KlepV2021 : ITF_OpenDichtKlep;
	KlepV2023 : ITF_OpenDichtKlep;
	KlepV2024 : ITF_OpenDichtKlep;
	
	SchuifV2013_AFO : ITF_Regelschuif;
	SchuifV2022_AFO : ITF_Regelschuif;
	
	SchuifV2013_DG : ITF_Regelschuif;
	SchuifV2022_DG : ITF_Regelschuif;

	Stand2013: SINT; //Moeten we van de regelingen krijgen
	Stand2022: SINT; //Moeten we van de regelingen krijgen
END_VAR

Stand2013 := main.Regelingen.RegelschuifStandV2013;
Stand2022 := main.Regelingen.RegelschuifStandV2022;
IF main.Regelingen.BestuurMode = E_Besturingsmodus.uitlaten THEN
	
	KlepV2012.Open();
	KlepV2021.Open();
	KlepV2023.Close();
	KlepV2024.Close();
	
	PompStatus11.PompGoTo(0);
	PompStatus21.PompGoTo(0);
	
	//Op het moment dat de terugmelding is gegeven dan:
	IF KlepV2012.StateKlep = E_OpenDichtKlepState.open AND KlepV2021.StateKlep = E_OpenDichtKlepState.open AND KlepV2023.StateKlep = E_OpenDichtKlepState.closed AND KlepV2024.StateKlep = E_OpenDichtKlepState.closed THEN		
		SchuifV2013_DG.RegelSchuifGoTo(Stand2013);
		
		IF ((SchuifV2013_AFO.ActueelPosition = Stand2013) OR (SchuifV2013_DG.ActueelPosition = Stand2013 ))THEN    
		SchuifV2022_DG.RegelSchuifGoTo(Stand2022);
	    END_IF
	END_IF
END_IF

//FB_Init is always available implicitly and it is used primarily for initialization.
//The return value is not evaluated. For a specific influence, you can also declare the
//methods explicitly and provide additional code there with the standard initialization
//code. You can evaluate the return value.
METHOD FB_Init: BOOL
VAR_INPUT
    bInitRetains: BOOL; // TRUE: the retain variables are initialized (reset warm / reset cold)
    bInCopyCode: BOOL;  // TRUE: the instance will be copied to the copy code afterward (online change)  
	OpenDichtKlepV2012: ITF_OpenDichtKlep;
	OpenDichtKlepV2021: ITF_OpenDichtKlep;
	OpenDichtKlepV2023: ITF_OpenDichtKlep;
	OpenDichtKlepV2024: ITF_OpenDichtKlep;
	
	V2013_DG: ITF_Regelschuif;
	V2022_DG: ITF_Regelschuif;
	
	V2013_AFO: ITF_Regelschuif;
	V2022_AFO: ITF_Regelschuif;
	
	Pomp2011: ITF_Pomp;
	Pomp2021: ITF_Pomp;
END_VAR
KlepV2012:= OpenDichtKlepV2012;
KlepV2021:= OpenDichtKlepV2021;
KlepV2023:= OpenDichtKlepV2023;
KlepV2024:= OpenDichtKlepV2024;

SchuifV2013_DG:= V2013_DG;
SchuifV2022_DG:= V2022_DG;

SchuifV2013_AFO:= V2013_AFO;
SchuifV2022_AFO:= V2022_AFO;

Pompstatus11:= Pomp2011;
Pompstatus21:= Pomp2021;
END_METHOD

END_FUNCTION_BLOCK

// ---- GlobalTextList.TcGTLO
TEXTLIST GlobalTextList
  7 = '%s'
  664 = 'actual percentage: %s'
  577 = 'ActueelToerental: %s'
  114 = 'AFO regelschuif test (V2013)'
  887 = 'AFO regelschuif test (V2022)'
  128 = 'analog out %s'
  781 = 'Auto'
  647 = 'Bedrijfstoestand %s'
  403 = 'Bedrijfstoestand: %s'
  441 = 'Bedrijftoestand: %s'
  497 = 'Closing'
  564 = 'dig in p2011'
  316 = 'Digital In 1'
  170 = 'Digital In 1 (close)'
  563 = 'Digital In 2'
  84 = 'Digital In 2 (open)'
  662 = 'Digital Out 1'
  792 = 'Digital Out 1 (off = closing, on = opening)'
  932 = 'DoelToerental: %s'
  547 = 'DoelToerentall: %s'
  359 = 'Feedback stand: %s'
  247 = 'InputSensor'
  249 = 'Manual'
  631 = 'Manual Close'
  416 = 'Manual Open'
  525 = 'Manualstand'
  513 = 'ManualStand'
  811 = 'Manualtoerental'
  702 = 'niet final'
  868 = 'Noodstop'
  59 = 'Off'
  591 = 'Ontluchtingskleppen'
  184 = 'Open/Dicht kleppen'
  164 = 'Opening'
  605 = 'Output'
  225 = 'P2011'
  113 = 'P2021'
  206 = 'P2099'
  991 = 'Position: %s'
  587 = 'pulse?'
  432 = 'Regelschuif'
  9 = 'set target margin: %s'
  542 = 'Standby'
  166 = 'standby'
  235 = 'Start'
  724 = 'Start '
  652 = 'Start proces '
  943 = 'State: %s'
  21 = 'Status: %s'
  610 = 'stop'
  992 = 'Stop'
  211 = 'Stop proces'
  980 = 'target percentage: %s'
  347 = 'Terugmelding'
  933 = 'TerugmeldingSensor'
  228 = 'Toerental SP (rpm)'
  493 = 'V2012'
  750 = 'V2012 Bedrijfstoestand: %s'
  859 = 'V2012 Mode: %s'
  69 = 'V2012 State: %s'
  826 = 'V2013_DG'
  322 = 'V2014'
  553 = 'V2021'
  755 = 'V2021 Bedrijfstoestand: %s'
  554 = 'V2021 State: %s'
  946 = 'V2022_DG'
  754 = 'V2023'
  181 = 'V2024'
  884 = 'V2025'
  533 = 'V2026'
  308 = 'Visvriendelijk'
END_TEXTLIST

// ---- VISUs/Visualization.TcVIS
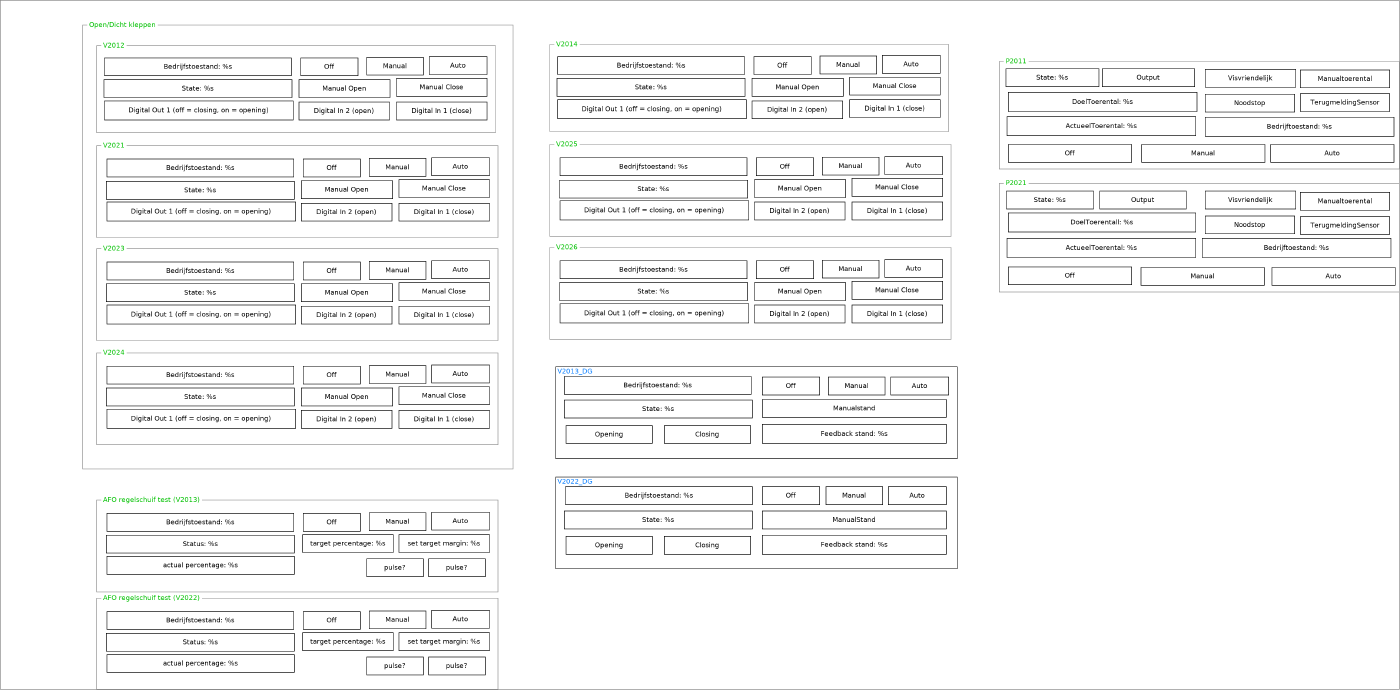
VISUALIZATION Visualization  // 2311x1139
    GroupBox (907,230 663x160), "V2025"
        RoundedRectangle (338,103 150x30), "Digital In 2 (open)", colour toggle: MAIN.digIn_V2025_2.internalState
            OnMouseDown: toggle MAIN.digIn_V2025_2.internalState
        RoundedRectangle (17,30 309x30), "Bedrijfstoestand: %s", text variable: MAIN.V2025.currentMode
        RoundedRectangle (450,29 94x30), "Manual"
            OnMouseDown: execute { MAIN.V2025.currentMode := E_Bedrijfstoestand.manual; }
        RoundedRectangle (553,28 96x30), "Auto"
            OnMouseDown: execute { MAIN.V2025.currentMode := E_Bedrijfstoestand.auto; }
        RoundedRectangle (17,101 312x32), "Digital Out 1 (off = closing, on = opening)", colour toggle: MAIN.digOut_V2025.internalState
        RoundedRectangle (338,66 151x30), "Manual Open"
            OnMouseDown: execute { MAIN.V2025.manOpen := TRUE; }
        RoundedRectangle (499,64 150x30), "Manual Close"
            OnMouseDown: execute { MAIN.V2025.manClose := TRUE; }
        RoundedRectangle (499,103 150x30), "Digital In 1 (close)", colour toggle: MAIN.digIn_V2025_1.internalState
            OnMouseDown: toggle MAIN.digIn_V2025_1.internalState
        RoundedRectangle (341,30 95x30), "Off"
            OnMouseDown: execute { MAIN.V2025.currentMode := E_Bedrijfstoestand.off; }
        RoundedRectangle (16,67 311x30), "State: %s", text variable: MAIN.V2025.currentState
    GroupBox (907,65 659x152), "V2014"
        RoundedRectangle (334,101 150x30), "Digital In 2 (open)", colour toggle: MAIN.digIn_V2014_2.internalState
            OnMouseDown: toggle MAIN.digIn_V2014_2.internalState
        RoundedRectangle (12,64 311x30), "State: %s", text variable: MAIN.V2014.currentState
        RoundedRectangle (13,28 309x30), "Bedrijfstoestand: %s", text variable: MAIN.V2014.currentMode
        RoundedRectangle (446,27 94x30), "Manual"
            OnMouseDown: execute { MAIN.V2014.currentMode := E_Bedrijfstoestand.manual; }
        RoundedRectangle (549,26 96x30), "Auto"
            OnMouseDown: execute { MAIN.V2014.currentMode := E_Bedrijfstoestand.auto; }
        RoundedRectangle (13,99 312x32), "Digital Out 1 (off = closing, on = opening)", colour toggle: MAIN.digOut_V2014.internalState
        RoundedRectangle (334,64 151x30), "Manual Open"
            OnMouseDown: execute { MAIN.V2014.manOpen := TRUE; }
        RoundedRectangle (495,62 150x30), "Manual Close"
            OnMouseDown: execute { MAIN.V2014.manClose := TRUE; }
        RoundedRectangle (495,99 150x30), "Digital In 1 (close)", colour toggle: MAIN.digIn_V2014_1.internalState
            OnMouseDown: toggle MAIN.digIn_V2014_1.internalState
        RoundedRectangle (337,28 95x30), "Off"
            OnMouseDown: execute { MAIN.V2014.currentMode := E_Bedrijfstoestand.off; }
    GroupBox (907,400 663x160), "V2026"
        RoundedRectangle (338,103 150x30), "Digital In 2 (open)", colour toggle: MAIN.digIn_V2026_2.internalState
            OnMouseDown: toggle MAIN.digIn_V2026_2.internalState
        RoundedRectangle (16,66 311x30), "State: %s", text variable: MAIN.V2026.currentState
        RoundedRectangle (17,30 309x30), "Bedrijfstoestand: %s", text variable: MAIN.V2026.currentMode
        RoundedRectangle (450,29 94x30), "Manual"
            OnMouseDown: execute { MAIN.V2026.currentMode := E_Bedrijfstoestand.manual; }
        RoundedRectangle (553,28 96x30), "Auto"
            OnMouseDown: execute { MAIN.V2026.currentMode := E_Bedrijfstoestand.auto; }
        RoundedRectangle (17,101 312x32), "Digital Out 1 (off = closing, on = opening)", colour toggle: MAIN.digOut_V2026.internalState
        RoundedRectangle (338,66 151x30), "Manual Open"
            OnMouseDown: execute { MAIN.V2026.manOpen := TRUE; }
        RoundedRectangle (499,64 150x30), "Manual Close"
            OnMouseDown: execute { MAIN.V2026.manClose := TRUE; }
        RoundedRectangle (499,103 150x30), "Digital In 1 (close)", colour toggle: MAIN.digIn_V2026_1.internalState
            OnMouseDown: toggle MAIN.digIn_V2026_1.internalState
        RoundedRectangle (341,30 95x30), "Off"
            OnMouseDown: execute { MAIN.V2026.currentMode := E_Bedrijfstoestand.off; }
    Group (136,33 711x741)
        GroupBox (23,199 663x160), "V2021"
            RoundedRectangle (338,103 150x30), "Digital In 2 (open)", colour toggle: MAIN.digIn_V2021_2.internalState
                OnMouseDown: toggle MAIN.digIn_V2021_2.internalState
            RoundedRectangle (17,30 309x30), "Bedrijfstoestand: %s", text variable: MAIN.V2021.currentMode
            RoundedRectangle (450,29 94x30), "Manual"
                OnMouseDown: execute { MAIN.V2021.currentMode := E_Bedrijfstoestand.manual; }
            RoundedRectangle (553,28 96x30), "Auto"
                OnMouseDown: execute { MAIN.V2021.currentMode := E_Bedrijfstoestand.auto; }
            RoundedRectangle (17,101 312x32), "Digital Out 1 (off = closing, on = opening)", colour toggle: MAIN.digOut_V2021.internalState
            RoundedRectangle (338,66 151x30), "Manual Open"
                OnMouseDown: execute { MAIN.V2021.manOpen := TRUE; }
            RoundedRectangle (499,64 150x30), "Manual Close"
                OnMouseDown: execute { MAIN.V2021.manClose := TRUE; }
            RoundedRectangle (499,103 150x30), "Digital In 1 (close)", colour toggle: MAIN.digIn_V2021_1.internalState
                OnMouseDown: toggle MAIN.digIn_V2021_1.internalState
            RoundedRectangle (341,30 95x30), "Off"
                OnMouseDown: execute { MAIN.V2021.currentMode := E_Bedrijfstoestand.off; }
            RoundedRectangle (16,67 311x30), "State: %s", text variable: MAIN.V2021.currentState
        GroupBox (23,34 659x152), "V2012"
            RoundedRectangle (334,101 150x30), "Digital In 2 (open)", colour toggle: MAIN.digIn_V2012_2.internalState
                OnMouseDown: toggle MAIN.digIn_V2012_2.internalState
            RoundedRectangle (12,64 311x30), "State: %s", text variable: MAIN.V2012.currentState
            RoundedRectangle (13,28 309x30), "Bedrijfstoestand: %s", text variable: MAIN.V2012.currentMode
            RoundedRectangle (446,27 94x30), "Manual"
                OnMouseDown: execute { MAIN.V2012.currentMode := E_Bedrijfstoestand.manual; }
            RoundedRectangle (549,26 96x30), "Auto"
                OnMouseDown: execute { MAIN.V2012.currentMode := E_Bedrijfstoestand.auto; }
            RoundedRectangle (13,99 312x32), "Digital Out 1 (off = closing, on = opening)", colour toggle: MAIN.digOut_V2012.internalState
            RoundedRectangle (334,64 151x30), "Manual Open"
                OnMouseDown: execute { MAIN.V2012.manOpen := TRUE; }
            RoundedRectangle (495,62 150x30), "Manual Close"
                OnMouseDown: execute { MAIN.V2012.manClose := TRUE; }
            RoundedRectangle (495,101 150x30), "Digital In 1 (close)", colour toggle: MAIN.digIn_V2012_1.internalState
                OnMouseDown: toggle MAIN.digIn_V2012_1.internalState
            RoundedRectangle (337,28 95x30), "Off"
                OnMouseDown: execute { MAIN.V2012.currentMode := E_Bedrijfstoestand.off; }
        GroupBox (23,369 663x160), "V2023"
            RoundedRectangle (338,103 150x30), "Digital In 2 (open)", colour toggle: MAIN.digIn_V2023_2.internalState
                OnMouseDown: toggle MAIN.digIn_V2023_2.internalState
            RoundedRectangle (16,66 311x30), "State: %s", text variable: MAIN.V2023.currentState
            RoundedRectangle (17,30 309x30), "Bedrijfstoestand: %s", text variable: MAIN.V2023.currentMode
            RoundedRectangle (450,29 94x30), "Manual"
                OnMouseDown: execute { MAIN.V2023.currentMode := E_Bedrijfstoestand.manual; }
            RoundedRectangle (553,28 96x30), "Auto"
                OnMouseDown: execute { MAIN.V2023.currentMode := E_Bedrijfstoestand.auto; }
            RoundedRectangle (17,101 312x32), "Digital Out 1 (off = closing, on = opening)", colour toggle: MAIN.digOut_V2023.internalState
            RoundedRectangle (338,66 151x30), "Manual Open"
                OnMouseDown: execute { MAIN.V2023.manOpen := TRUE; }
            RoundedRectangle (499,64 150x30), "Manual Close"
                OnMouseDown: execute { MAIN.V2023.manClose := TRUE; }
            RoundedRectangle (499,103 150x30), "Digital In 1 (close)", colour toggle: MAIN.digIn_V2023_1.internalState
                OnMouseDown: toggle MAIN.digIn_V2023_1.internalState
            RoundedRectangle (341,30 95x30), "Off"
                OnMouseDown: execute { MAIN.V2023.currentMode := E_Bedrijfstoestand.off; }
        GroupBox (23,541 663x160), "V2024"
            RoundedRectangle (338,103 150x30), "Digital In 2 (open)", colour toggle: MAIN.digIn_V2024_2.internalState
                OnMouseDown: toggle MAIN.digIn_V2024_2.internalState
            RoundedRectangle (16,66 311x30), "State: %s", text variable: MAIN.V2024.currentState
            RoundedRectangle (17,30 309x30), "Bedrijfstoestand: %s", text variable: MAIN.V2024.currentMode
            RoundedRectangle (450,29 94x30), "Manual"
                OnMouseDown: execute { MAIN.V2024.currentMode := E_Bedrijfstoestand.manual; }
            RoundedRectangle (553,28 96x30), "Auto"
                OnMouseDown: execute { MAIN.V2024.currentMode := E_Bedrijfstoestand.auto; }
            RoundedRectangle (17,101 312x32), "Digital Out 1 (off = closing, on = opening)", colour toggle: MAIN.digOut_V2024.internalState
            RoundedRectangle (338,66 151x30), "Manual Open"
                OnMouseDown: execute { MAIN.V2024.manOpen := TRUE; }
            RoundedRectangle (499,64 150x30), "Manual Close"
                OnMouseDown: execute { MAIN.V2024.manClose := TRUE; }
            RoundedRectangle (499,103 150x30), "Digital In 1 (close)", colour toggle: MAIN.digIn_V2024_1.internalState
                OnMouseDown: toggle MAIN.digIn_V2024_1.internalState
            RoundedRectangle (341,30 95x30), "Off"
                OnMouseDown: execute { MAIN.V2024.currentMode := E_Bedrijfstoestand.off; }
        GroupBox (0,0 711x741), "Open/Dicht kleppen"
    GroupBox (1649,294 661x188), "P2021"
        RoundedRectangle (13,99 312x32), "ActueelToerental: %s", text variable: MAIN.AnaoutP2021.internalState
        RoundedRectangle (340,62 148x30), "Noodstop"
            OnMouseDown: execute { MAIN.P2021.noodstop := true; }
        RoundedRectangle (166,21 143x30), "Output", colour toggle: MAIN.digoutP2021.internalState
        RoundedRectangle (12,21 144x30), "State: %s", text variable: MAIN.P2021.InternalState
        RoundedRectangle (340,21 150x30), "Visvriendelijk", colour toggle: MAIN.P2021.visvriendelijkactief
            OnMouseClick: execute {  }
            OnMouseClick: toggle main.P2021.visvriendelijkactief
        RoundedRectangle (497,63 148x30), "TerugmeldingSensor", colour toggle: MAIN.diginP2021.internalState
            OnMouseDown: execute {  }
            OnMouseDown: toggle MAIN.diginP2021.internalState
        RoundedRectangle (497,23 148x30), "Manualtoerental"
            OnMouseDown: write MAIN.ManToerental2021 via VisuDialogs.Numpad
        RoundedRectangle (15,146 204x30), "Off"
            OnMouseDown: execute { Main.P2021.bedrijftoestand := E_bedrijfstoestand.off; }
        RoundedRectangle (234,147 204x30), "Manual"
            OnMouseDown: execute { Main.P2021.bedrijftoestand := E_bedrijfstoestand.manual; }
        RoundedRectangle (450,147 204x30), "Auto"
            OnMouseDown: execute { Main.P2021.bedrijftoestand := E_bedrijfstoestand.auto; }
        RoundedRectangle (335,99 312x32), "Bedrijftoestand: %s", text variable: MAIN.P2021.Bedrijftoestand
        RoundedRectangle (15,57 310x32), "DoelToerentall: %s", text variable: MAIN.P2021.globaaldoeltoerental
    GroupBox (1649,93 662x186), "P2011"
        RoundedRectangle (13,99 312x32), "ActueelToerental: %s", text variable: MAIN.AnaoutP2011.internalState
        RoundedRectangle (340,62 148x30), "Noodstop"
            OnMouseDown: execute { MAIN.P2011.noodstop := true; }
        RoundedRectangle (170,20 153x30), "Output", colour toggle: MAIN.digoutP2011.internalState
        RoundedRectangle (11,20 154x30), "State: %s", text variable: MAIN.P2011.InternalState
        RoundedRectangle (340,21 150x30), "Visvriendelijk", colour toggle: MAIN.P2011.visvriendelijkactief
            OnMouseClick: execute {  }
            OnMouseClick: toggle main.P2011.visvriendelijkactief
        RoundedRectangle (497,61 148x30), "TerugmeldingSensor", colour toggle: MAIN.diginP2011.internalState
            OnMouseDown: execute {  }
            OnMouseDown: toggle MAIN.diginP2011.internalState
        RoundedRectangle (497,22 148x30), "Manualtoerental"
            OnMouseDown: write MAIN.ManToerental2011 via VisuDialogs.Numpad
        RoundedRectangle (340,100 312x32), "Bedrijftoestand: %s", text variable: MAIN.P2011.Bedrijftoestand
        RoundedRectangle (15,145 204x30), "Off"
            OnMouseDown: execute { main.P2011.bedrijftoestand := E_bedrijfstoestand.off; }
        RoundedRectangle (235,145 204x30), "Manual"
            OnMouseDown: execute { Main.P2011.bedrijftoestand := E_bedrijfstoestand.manual; }
        RoundedRectangle (448,145 204x30), "Auto"
            OnMouseDown: execute { Main.P2011.bedrijftoestand := E_bedrijfstoestand.auto; }
        RoundedRectangle (15,59 312x32), "DoelToerental: %s", text variable: MAIN.P2011.globaaldoeltoerental
    Rectangle (917,605 663x152), "V2013_DG"
    RoundedRectangle (931,621 309x30), "Bedrijfstoestand: %s", text variable: MAIN.V2013_DG.CurrentMode
    RoundedRectangle (1258,622 95x30), "Off"
        OnMouseDown: execute { MAIN.V2013_DG.CurrentMode:= E_Bedrijfstoestand.off; }
    RoundedRectangle (1367,622 94x30), "Manual"
        OnMouseDown: execute { MAIN.V2013_DG.currentMode := E_Bedrijfstoestand.manual; }
    RoundedRectangle (1470,622 96x30), "Auto"
        OnMouseDown: execute { MAIN.V2013_DG.currentMode := E_Bedrijfstoestand.auto; }
    RoundedRectangle (931,660 311x30), "State: %s", text variable: MAIN.V2013_DG.currentState
    Rectangle (917,787 663x152), "V2022_DG"
    RoundedRectangle (933,803 309x30), "Bedrijfstoestand: %s", text variable: MAIN.V2022_DG.CurrentMode
    RoundedRectangle (931,843 311x30), "State: %s", text variable: MAIN.V2022_DG.currentState
    RoundedRectangle (1258,803 95x30), "Off"
        OnMouseDown: execute { MAIN.V2022_DG.CurrentMode:= E_Bedrijfstoestand.off; }
    RoundedRectangle (1363,803 94x30), "Manual"
        OnMouseDown: execute { MAIN.V2022_DG.currentMode := E_Bedrijfstoestand.manual; }
    RoundedRectangle (1466,803 96x30), "Auto"
        OnMouseDown: execute { MAIN.V2022_DG.currentMode := E_Bedrijfstoestand.auto; }
    RoundedRectangle (1258,659 304x30), "Manualstand"
        OnMouseDown: write MAIN.ManKlepstand2013_DG via VisuDialogs.Numpad
    RoundedRectangle (1258,843 304x30), "ManualStand"
        OnMouseDown: write MAIN.ManKlepstand2022_DG via VisuDialogs.Numpad
    RoundedRectangle (1258,700 304x32), "Feedback stand: %s", text variable: MAIN.V2013_DG.feedbackposition
    RoundedRectangle (1258,883 304x32), "Feedback stand: %s", text variable: MAIN.V2022_DG.feedbackposition
    RoundedRectangle (934,885 143x30), "Opening", colour toggle: MAIN.OutOpeningV2022.internalState
    RoundedRectangle (1096,885 143x30), "Closing", colour toggle: MAIN.OutClosingV2022.internalState
    RoundedRectangle (934,702 143x30), "Opening", colour toggle: MAIN.OutOpeningV2013.internalState
    RoundedRectangle (1096,702 143x30), "Closing", colour toggle: MAIN.OutClosingV2013.internalState
    GroupBox (159,817 663x160), "AFO regelschuif test (V2013)", tooltip "niet final"
        RoundedRectangle (16,66 311x30), "Status: %s", text variable: MAIN.V2013_AFO.currentState
        RoundedRectangle (17,30 309x30), "Bedrijfstoestand: %s", text variable: MAIN.V2013_AFO.currentMode
        RoundedRectangle (450,29 94x30), "Manual"
            OnMouseDown: execute { MAIN.V2013_afo.currentMode := E_Bedrijfstoestand.manual; }
        RoundedRectangle (553,28 96x30), "Auto"
            OnMouseDown: execute { MAIN.V2013_afo.currentMode := E_Bedrijfstoestand.auto; }
        RoundedRectangle (341,30 95x30), "Off"
            OnMouseDown: execute { MAIN.V2013_afo.currentMode := E_Bedrijfstoestand.off; }
        RoundedRectangle (499,65 150x30), "set target margin: %s", text variable: MAIN.V2013_AFO.regelschuifMargin
            OnMouseDown: write the text variable via Default, min 0, max 100
        RoundedRectangle (17,101 310x30), "actual percentage: %s", text variable: MAIN.AnaInV2013.internalState
            OnMouseDown: write the text variable via Default, min 0, max 100
        RoundedRectangle (446,105 94x30), "pulse?", colour toggle: MAIN.digOutClosingV2013.internalState
    RoundedRectangle (499,882 150x30), "target percentage: %s", text variable: MAIN.AFOTarget
        OnMouseDown: write the text variable via Default, min 0, max 100
    RoundedRectangle (707,922 94x30), "pulse?", colour toggle: MAIN.digOutOpeningV2013.internalState
    GroupBox (159,979 663x160), "AFO regelschuif test (V2022)", tooltip "niet final"
        RoundedRectangle (16,66 311x30), "Status: %s", text variable: MAIN.V2022_AFO.currentState
        RoundedRectangle (17,30 309x30), "Bedrijfstoestand: %s", text variable: MAIN.V2022_AFO.currentMode
        RoundedRectangle (450,29 94x30), "Manual"
            OnMouseDown: execute { MAIN.V2022_afo.currentMode := E_Bedrijfstoestand.manual; }
        RoundedRectangle (553,28 96x30), "Auto"
            OnMouseDown: execute { MAIN.V2022_afo.currentMode := E_Bedrijfstoestand.auto; }
        RoundedRectangle (341,30 95x30), "Off"
            OnMouseDown: execute { MAIN.V2022_afo.currentMode := E_Bedrijfstoestand.off; }
        RoundedRectangle (499,65 150x30), "set target margin: %s", text variable: MAIN.V2022_AFO.regelschuifMargin
            OnMouseDown: write the text variable via Default, min 0, max 100
        RoundedRectangle (17,101 310x30), "actual percentage: %s", text variable: MAIN.AnaInV2022.internalState
            OnMouseDown: write the text variable via Default, min 0, max 100
        RoundedRectangle (446,105 94x30), "pulse?", colour toggle: MAIN.digOutClosingV2022.internalState
    RoundedRectangle (499,1044 150x30), "target percentage: %s", text variable: MAIN.AFOTarget2
        OnMouseDown: write the text variable via Default, min 0, max 100
    RoundedRectangle (707,1084 94x30), "pulse?", colour toggle: MAIN.digOutOpeningV2022.internalState
END_VISUALIZATION
